// TIA Portal V21 export
VAR_GLOBAL   // PLC tag table "KAllAnalogica"
END_VAR
VAR_GLOBAL CONSTANT   // user constants
   KAllAnalog_Maxi : Int := 1;   // Maximale Schwelle ausgelöst / Maximum threshold reached / Umbral máximo intervenido / Seuil maximum intervenu / Soglia massima intervenuta
   KAllAnalog_IntMax : Int := 2;   // Maximale Zwischenschwelle ausgelöst / Maximum intermediate threshold intervened / Umbral intermedio máximo intervenido / Seuil intermédiaire maximal intervenu / Soglia intermedia massima intervenuta
   KAllAnalog_IntMin : Int := 3;   // Eingriffsminimaler Zwischenschwellenwert / Minimum intermediate threshold intervened / Umbral intermedio mínimo intervenido / Seuil intermédiaire minimal intervenu / Soglia intermedia minima intervenuta
   KAllAnalog_Mini : Int := 4;   // Eingriffsmindestschwelle / Minimum threshold intervened / Umbral mínimo intervenido / Seuil minimum intervenu / Soglia minima intervenuta
   KAllAnalog_OutOfRange : Int := 5;   // Sonde außerhalb des Messbereichs / Out of range of measurement / Sonda fuera del rango de medición / Sonde en dehors de la plage de mesure / Sonda fuori dal range di misurazione
   KALLAnalogica_06 : Int := 6;
   KALLAnalogica_07 : Int := 7;
   KALLAnalogica_08 : Int := 8;
   KALLAnalogica_09 : Int := 9;
   KALLAnalogica_10 : Int := 10;
   KALLAnalogica_11 : Int := 11;
   KALLAnalogica_12 : Int := 12;
   KALLAnalogica_13 : Int := 13;
   KALLAnalogica_14 : Int := 14;
   KALLAnalogica_15 : Int := 15;
   KALLAnalogica_16 : Int := 16;
END_VAR
